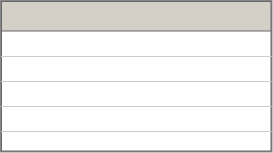
VISUALIZATION _VisuAddressSelector  // 273x153
    Table (1,1 270x150), data array: ComGVL._glAddressNameTable
        p3854506369: ComGVL._glAddressNameTable[INDEX]
        p2232123230: Station Address
        p1137915858: ComGVL._glAddressSelectionIndex
END_VISUALIZATION

(* stored: Version 1.1.0.1, ProductVersion 3.1.4024.2
   Visu _VisuAddressSelector: Id {6e76abbd-8818-407d-9a5e-c52b73c6b4d0} *)
